FUNCTION_BLOCK FB_ESCcommunication
VAR_INPUT
	
senddata : STRING;

END_VAR

VAR_IN_OUT
	TxBuffer	: ComBuffer;
	RxBuffer	: ComBuffer;
END_VAR
VAR_OUTPUT
	bReceiveError	: BOOL;
	eReceiveErrorID	: ComError_t;
END_VAR
VAR
	Timer		: TON := (PT:=T#1S);
	fbSend		: SendString;
	bSendBusy	: BOOL;
	eSendErrorID: ComError_t;

	fbReceive		: ReceiveString;
	sReceivedString	: STRING;
	sLastReceivedString: STRING;
	bStringReceived	: BOOL;
	bReceiveBusy	: BOOL;
	bReceiveTimeout	: BOOL;
	nReceiveCounter	: UDINT;
END_VAR

Timer(IN:=TRUE);
IF Timer.Q OR fbSend.Busy THEN
	Timer(IN:=FALSE); (* reset timer *)
	fbSend(	SendString:= senddata,
			TXbuffer:= TxBuffer,
			Busy=> bSendBusy,
			Error=> );
	IF fbSend.Error <> COMERROR_NOERROR THEN
		eSendErrorID := fbSend.Error;
	END_IF
END_IF

fbReceive(
	Prefix:= '',
	Suffix:= '',
	Timeout:= T#1s,
	ReceivedString:= sReceivedString,
	RXbuffer:= RxBuffer,
	StringReceived=> bStringReceived,
	Busy=> bReceiveBusy,
	Error=> ,
	RxTimeout=> bReceiveTimeout );
IF fbReceive.Error <> COMERROR_NOERROR THEN
	eReceiveErrorID := fbReceive.Error;
END_IF
IF bStringReceived THEN
	nReceiveCounter := nReceiveCounter + 1;
	sLastReceivedString := sReceivedString;
END_IF

END_FUNCTION_BLOCK

(* stored: Version 1.1.0.1, ProductVersion 3.1.4024.13
   POU FB_ESCcommunication: Id {f8d71dd6-03ac-4bbb-83ef-f6182c2a2131}, SpecialFunc None *)
